# EPICS substitutions: db/ecmciPOS4808.substitutions
file ecmcEcSlave.template
{
    pattern {}
            {}
}

file ecmcIPOSXXXX_DRV.template
{
	pattern {LINR,    ESLO,   EOFF,   EGU,        PREC, LOW, LOLO, HIGH, HIHI, HYST, LLSV,       LSV,        HSV,        HHSV      }
		{"SLOPE", 1,      0,      "Raw",      0,    0,   0,    0,    0,    0,    "NO_ALARM", "NO_ALARM", "NO_ALARM", "NO_ALARM"}
}

file ecmcIPOSXXXX_ENC.template
{
	pattern {LINR,    ESLO,   EOFF,   EGU,        PREC, LOW, LOLO, HIGH, HIHI, HYST, LLSV,       LSV,        HSV,        HHSV      }
		{"SLOPE", 1,      0,      "Raw",      0,    0,   0,    0,    0,    0,    "NO_ALARM", "NO_ALARM", "NO_ALARM", "NO_ALARM"}
}

file ecmcIPOSXXXX_AUX.template
{
	pattern {CURRESLO}
    		{6.105e-4}
}
